INTERFACE I_KeyValueCollection EXTENDS I_Enumerable, I_Disposable, I_EventEmitter

END_INTERFACE

(* stored: Version 1.1.0.1, ProductVersion 3.1.4024.12
   Itf I_KeyValueCollection: Id {8afa0049-808e-42a5-a811-87c8f4a10e9f} *)
